{attribute 'no_explicit_call' := 'NoCommand is a CLASS and must be accessed using methods or properties'}
FUNCTION_BLOCK NoCommand IMPLEMENTS I_Command
VAR
END_VAR
/// Command that does nothing for base initialization

METHOD Execute
END_METHOD

END_FUNCTION_BLOCK

(* stored: Version 1.1.0.1, ProductVersion 3.1.4024.12
   POU NoCommand: Id {a401e31b-9139-4a9e-b5cd-f1c627427aee}, SpecialFunc None
   Method Execute: Id {6d87fd1e-6241-474b-a0ec-b5689361a963} *)
